PROGRAM LOAD_NG
VAR
	DELAY: TON;
END_VAR

IF NOT SORTER_VAR.I_NG_TRANSFER_AT_BACK THEN
	SORTER_VAR.O_NG_DATA_OUTPUT2:=TRUE;
ELSE
	SORTER_VAR.O_NG_DATA_OUTPUT2:=FALSE;
END_IF

END_PROGRAM

(* stored: Version 1.1.0.1, ProductVersion 3.1.4020.12
   POU LOAD_NG: Id {2f23b999-c3ff-402f-a894-b44e03b27e70}, SpecialFunc None *)
